FUNCTION_BLOCK EcMasterGetDeviceCRC IMPLEMENTS IEcTask
VAR_INPUT
END_VAR
VAR_OUTPUT
END_VAR
VAR
	iState : INT;
	getDeviceCRC : Tc2_EtherCAT.FB_EcGetSlaveCrcErrorEx;
	_execute: BOOL;
	_done: BOOL;
	_busy: BOOL;
	_error: BOOL;
	_netId: AMSNETID;
END_VAR

CASE iState OF
	0:
		IF _execute THEN
			_done := FALSE;
			_busy := TRUE;
			_error := FALSE;
			getDeviceCRC.bExecute := TRUE;
			IF getDeviceCRC.bBusy THEN
				iState := 10;
				_execute := false;
			END_IF
		END_IF
	10:
		IF NOT getDeviceCRC.bBusy THEN
			IF NOT getDeviceCRC.bError THEN
				_done := TRUE;
			ELSE
				_error := TRUE;
			END_IF
			_busy := FALSE;
			getDeviceCRC.bExecute := FALSE;
			iState := 0;
		END_IF
END_CASE

getDeviceCRC(sNetId := Tc2_System.F_CreateAmsNetId(nIds := NetId));

{warning 'add method implementation '}
METHOD Abort : BOOL
getDeviceCRC.bExecute := FALSE;
_busy := FALSE;
_execute := FALSE;
Abort := TRUE;
iState := 0;
END_METHOD

{warning 'add property implementation'}
PROPERTY Busy : BOOL
GET
Busy := _busy;
END_GET
END_PROPERTY

PROPERTY DeviceAddr : uint
GET
DeviceAddr := getDeviceCRC.nSlaveAddr;
END_GET
SET
getDeviceCRC.nSlaveAddr := DeviceAddr;
END_SET
END_PROPERTY

PROPERTY DeviceCRC :  ST_EcCrcErrorEx
GET
DeviceCRC := getDeviceCRC.crcError;
END_GET
END_PROPERTY

{warning 'add property implementation'}
PROPERTY Done : BOOL
GET
Done := _done;
END_GET
END_PROPERTY

{warning 'add property implementation'}
PROPERTY Error : BOOL
GET
Error := _error;
END_GET
END_PROPERTY

{warning 'add method implementation '}
METHOD Execute : BOOL
IF NOT getDeviceCRC.bBusy THEN
	Execute := _execute := true;
END_IF
END_METHOD

{warning 'add property implementation'}
PROPERTY NetID : amsnetid
GET
NetID := _netId;
END_GET
SET
_netId := NetID;
END_SET
END_PROPERTY

END_FUNCTION_BLOCK

(* stored: Version 1.1.0.1, ProductVersion 3.1.4024.11
   POU EcMasterGetDeviceCRC: Id {2fe6c277-45c7-44ed-8725-6c8ed34fb399}, SpecialFunc None
   Method Abort: Id {f668e62a-1212-469d-8620-6274a6ff43fc}
   Property Busy: Id {ec61659d-4874-4473-ab1d-464cc4fbd5e3}
   Get Get: Id {1b91271c-4fa1-4b00-a7f4-e997e6f4b77e}
   Property DeviceAddr: Id {80b0df27-a43a-4fd8-86a2-6c73d6ff4483}
   Get Get: Id {291fc0c5-b305-46e5-add6-48d60348e373}
   Set Set: Id {68b97ca7-9867-44bf-8fe4-de13d96b439e}
   Property DeviceCRC: Id {332b4dca-4091-4557-9722-035187b3a5ff}
   Get Get: Id {9d5395e1-7e65-45ac-aa7c-ac987038081a}
   Property Done: Id {b9dbe9b2-e782-4383-b3b9-59408f19494b}
   Get Get: Id {a7b6fd00-89c1-43dc-8eac-af6dc313841b}
   Property Error: Id {32380371-432a-41e7-8535-1947b40047b9}
   Get Get: Id {c94de90c-5bb0-45fe-bd3b-b1dfb7e7729c}
   Method Execute: Id {4100fa81-cd09-4d6c-9799-eca9e4d7defa}
   Property NetID: Id {ea13d162-d47e-4fb2-813e-07ae1c2b7e9f}
   Get Get: Id {29241eeb-776b-4863-acb2-12d489c1d2d1}
   Set Set: Id {f1bc0a40-fd6e-4eea-a3f1-0e551472ac26} *)
